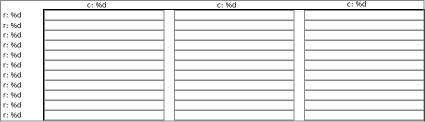
VISUALIZATION _VISU_DefGridTable  // 425x122
VAR_IN_OUT
	m_Inst : FB_ImageDeformation;
  m_row_start : UDINT;
  m_col_start : UDINT;
END_VAR
    Rectangle (43,9 382x112)
    Frame (44,10 120x10)
        shows _VISU_GridPointView(m_Inst := m_Inst._sDefGridPoints[0+m_col_start, 0+m_row_start])
    Frame (44,20 120x10)
        shows _VISU_GridPointView(m_Inst := m_Inst._sDefGridPoints[0+m_col_start, 1+m_row_start])
    Frame (44,30 120x10)
        shows _VISU_GridPointView(m_Inst := m_Inst._sDefGridPoints[0+m_col_start, 2+m_row_start])
    Frame (44,40 120x10)
        shows _VISU_GridPointView(m_Inst := m_Inst._sDefGridPoints[0+m_col_start, 3+m_row_start])
    Frame (44,50 120x10)
        shows _VISU_GridPointView(m_Inst := m_Inst._sDefGridPoints[0+m_col_start, 4+m_row_start])
    Frame (44,60 120x10)
        shows _VISU_GridPointView(m_Inst := m_Inst._sDefGridPoints[0+m_col_start, 5+m_row_start])
    Frame (44,70 120x10)
        shows _VISU_GridPointView(m_Inst := m_Inst._sDefGridPoints[0+m_col_start, 6+m_row_start])
    Frame (44,80 120x10)
        shows _VISU_GridPointView(m_Inst := m_Inst._sDefGridPoints[0+m_col_start, 7+m_row_start])
    Frame (44,90 120x10)
        shows _VISU_GridPointView(m_Inst := m_Inst._sDefGridPoints[0+m_col_start, 8+m_row_start])
    Frame (44,100 120x10)
        shows _VISU_GridPointView(m_Inst := m_Inst._sDefGridPoints[0+m_col_start, 9+m_row_start])
    Frame (44,110 120x10)
        shows _VISU_GridPointView(m_Inst := m_Inst._sDefGridPoints[0+m_col_start, 10+m_row_start])
    Frame (174,10 120x10)
        shows _VISU_GridPointView(m_Inst := m_Inst._sDefGridPoints[1+m_col_start, 0+m_row_start])
    Frame (174,20 120x10)
        shows _VISU_GridPointView(m_Inst := m_Inst._sDefGridPoints[1+m_col_start, 1+m_row_start])
    Frame (174,30 120x10)
        shows _VISU_GridPointView(m_Inst := m_Inst._sDefGridPoints[1+m_col_start, 2+m_row_start])
    Frame (174,40 120x10)
        shows _VISU_GridPointView(m_Inst := m_Inst._sDefGridPoints[1+m_col_start, 3+m_row_start])
    Frame (174,50 120x10)
        shows _VISU_GridPointView(m_Inst := m_Inst._sDefGridPoints[1+m_col_start, 4+m_row_start])
    Frame (174,60 120x10)
        shows _VISU_GridPointView(m_Inst := m_Inst._sDefGridPoints[1+m_col_start, 5+m_row_start])
    Frame (174,70 120x10)
        shows _VISU_GridPointView(m_Inst := m_Inst._sDefGridPoints[1+m_col_start, 6+m_row_start])
    Frame (174,80 120x10)
        shows _VISU_GridPointView(m_Inst := m_Inst._sDefGridPoints[1+m_col_start, 7+m_row_start])
    Frame (174,90 120x10)
        shows _VISU_GridPointView(m_Inst := m_Inst._sDefGridPoints[1+m_col_start, 8+m_row_start])
    Frame (174,100 120x10)
        shows _VISU_GridPointView(m_Inst := m_Inst._sDefGridPoints[1+m_col_start, 9+m_row_start])
    Frame (174,110 120x10)
        shows _VISU_GridPointView(m_Inst := m_Inst._sDefGridPoints[1+m_col_start, 10+m_row_start])
    Frame (304,10 120x10)
        shows _VISU_GridPointView(m_Inst := m_Inst._sDefGridPoints[2+m_col_start, 0+m_row_start])
    Frame (304,20 120x10)
        shows _VISU_GridPointView(m_Inst := m_Inst._sDefGridPoints[2+m_col_start, 1+m_row_start])
    Frame (304,30 120x10)
        shows _VISU_GridPointView(m_Inst := m_Inst._sDefGridPoints[2+m_col_start, 2+m_row_start])
    Frame (304,40 120x10)
        shows _VISU_GridPointView(m_Inst := m_Inst._sDefGridPoints[2+m_col_start, 3+m_row_start])
    Frame (304,50 120x10)
        shows _VISU_GridPointView(m_Inst := m_Inst._sDefGridPoints[2+m_col_start, 4+m_row_start])
    Frame (304,60 120x10)
        shows _VISU_GridPointView(m_Inst := m_Inst._sDefGridPoints[2+m_col_start, 5+m_row_start])
    Frame (304,70 120x10)
        shows _VISU_GridPointView(m_Inst := m_Inst._sDefGridPoints[2+m_col_start, 6+m_row_start])
    Frame (304,80 120x10)
        shows _VISU_GridPointView(m_Inst := m_Inst._sDefGridPoints[2+m_col_start, 7+m_row_start])
    Frame (304,90 120x10)
        shows _VISU_GridPointView(m_Inst := m_Inst._sDefGridPoints[2+m_col_start, 8+m_row_start])
    Frame (304,100 120x10)
        shows _VISU_GridPointView(m_Inst := m_Inst._sDefGridPoints[2+m_col_start, 9+m_row_start])
    Frame (304,110 120x10)
        shows _VISU_GridPointView(m_Inst := m_Inst._sDefGridPoints[2+m_col_start, 10+m_row_start])
    Rectangle (84,0 40x10), "c: %d", text variable: m_col_start
    Rectangle (214,0 40x10), "c: %d", text variable: m_col_start+1
    Rectangle (344,-1 40x10), "c: %d", text variable: m_col_start+2
    Rectangle (0,10 40x10), "r: %d", text variable: m_row_start
    Rectangle (0,20 40x11), "r: %d", text variable: m_row_start+1
    Rectangle (0,30 40x10), "r: %d", text variable: m_row_start+2
    Rectangle (0,40 40x10), "r: %d", text variable: m_row_start+3
    Rectangle (0,50 40x10), "r: %d", text variable: m_row_start+4
    Rectangle (0,60 40x10), "r: %d", text variable: m_row_start+5
    Rectangle (0,70 40x10), "r: %d", text variable: m_row_start+6
    Rectangle (0,80 40x10), "r: %d", text variable: m_row_start+7
    Rectangle (0,90 40x10), "r: %d", text variable: m_row_start+8
    Rectangle (0,100 40x10), "r: %d", text variable: m_row_start+9
    Rectangle (0,110 40x10), "r: %d", text variable: m_row_start+10
END_VISUALIZATION

(* stored: Version 1.1.0.1, ProductVersion 3.1.4024.3
   Visu _VISU_DefGridTable: Id {b6a9ffe9-c4ee-44c8-ad58-d26329db8e3e} *)
